{attribute 'GeneratedUsingTerminal: EK1122-0000-0018'}
{attribute addProperty BoxType "EK1122-0000-0018"}
{attribute addProperty Id "Term_11_EK1100Term_11_EK1100_B6553301142Term_18_EK1100Term_18_EK1100_249FE75772"}
{attribute addProperty CRC "3147807716"}
{attribute addProperty Size "214"}
TYPE Term_10_EK1122_BB9FBBE4 EXTENDS EK1122_1FC0878B :
STRUCT
	{attribute addProperty Name "Term 11 (EK1100)"}
	{attribute addProperty PreviousPort "Term 10 (EK1122) : D"}
	Term_11_EK1100 : Term_11_EK1100_B6553301;
	{attribute addProperty Name "Term 18 (EK1100)"}
	{attribute addProperty PreviousPort "Term 17 (EK1110) : B"}
	Term_18_EK1100 : Term_18_EK1100_249FE757;
END_STRUCT
END_TYPE

(* stored: Version 1.2.0.0, ProductVersion 3.1.4024.9
   DUT Term_10_EK1122_BB9FBBE4: Id {9cd0a634-f41d-06a2-336a-1a8dac19e3f7} *)
